(* Schneider Machine Expert - Basic project automat_biscuiti, file version 2.6.0.0 *)
(* ProjectInformations: Name=New project *)

HARDWARE
  Cpu 0: TM221M16R/G
  ModuleExtensionObject 0: TM3AM6/G
  ModuleExtensionObject 1: TM3AI8/G
  EthernetConfiguration: NetworkName=M221, IpAllocationMode=FixedAddress, IpAddress=0.0.0.0, SubnetMask=0.0.0.0
  SerialLineConfiguration: Baud=Baud19200, Parity=ParityEven, DataBits=DataBits8, StopBits=StopBits1, PhysicalMedium=PhysicalMediumRs485, TransmissionMode=TransmissionModeModbusRtu, SlaveId=1, Addressing=SlaveAddressing
  MastTask: UsePeriodScanMode=false, PeriodScan=100
  FastTask: Period=255
  CpuBehavior: StartingMode=StartAsPreviousState, AutoSaveRamOnEeprom=true, WatchdogPeriod=250

SYMBOLS  (address, symbol, comment, settings)
  %TM0        "Se pregatesc biscuitii"  [Preset=5, Base=OneSecond]
  %I0.0       "Faina fara gluten"
  %I0.1       "Faina integrala"
  %I0.2       "Lapte"
  %I0.3       "Lapte de soia"
  %I0.4       "Lapte de migdale"
  %I0.5       "Ou"
  %I0.6       "Inlocuitor ou"
  %I0.7       "Automat pornit"
  %Q0.0       "Faina fara gluten"
  %Q0.1       "Faina integrala"
  %Q0.2       "Lapte"
  %Q0.3       "Lapte de soia"
  %Q0.4       "Automat pornit - introduceti 15 lei"
  %Q0.5       "Ou"
  %Q0.6       "Inlocuitor ou"
  %Q0.7       "Cutie biscuiti servita"
  %IW0.0      [Type=Type_0_10V, Scope=Scope_Normal, Minimum=0, Maximum=1000]
  %IW1.1      [Type=Type_NotUsed, Scope=Scope_NotUsed, Minimum=0, Maximum=0]

POU New POU
  (* SectionNumber=1 *)

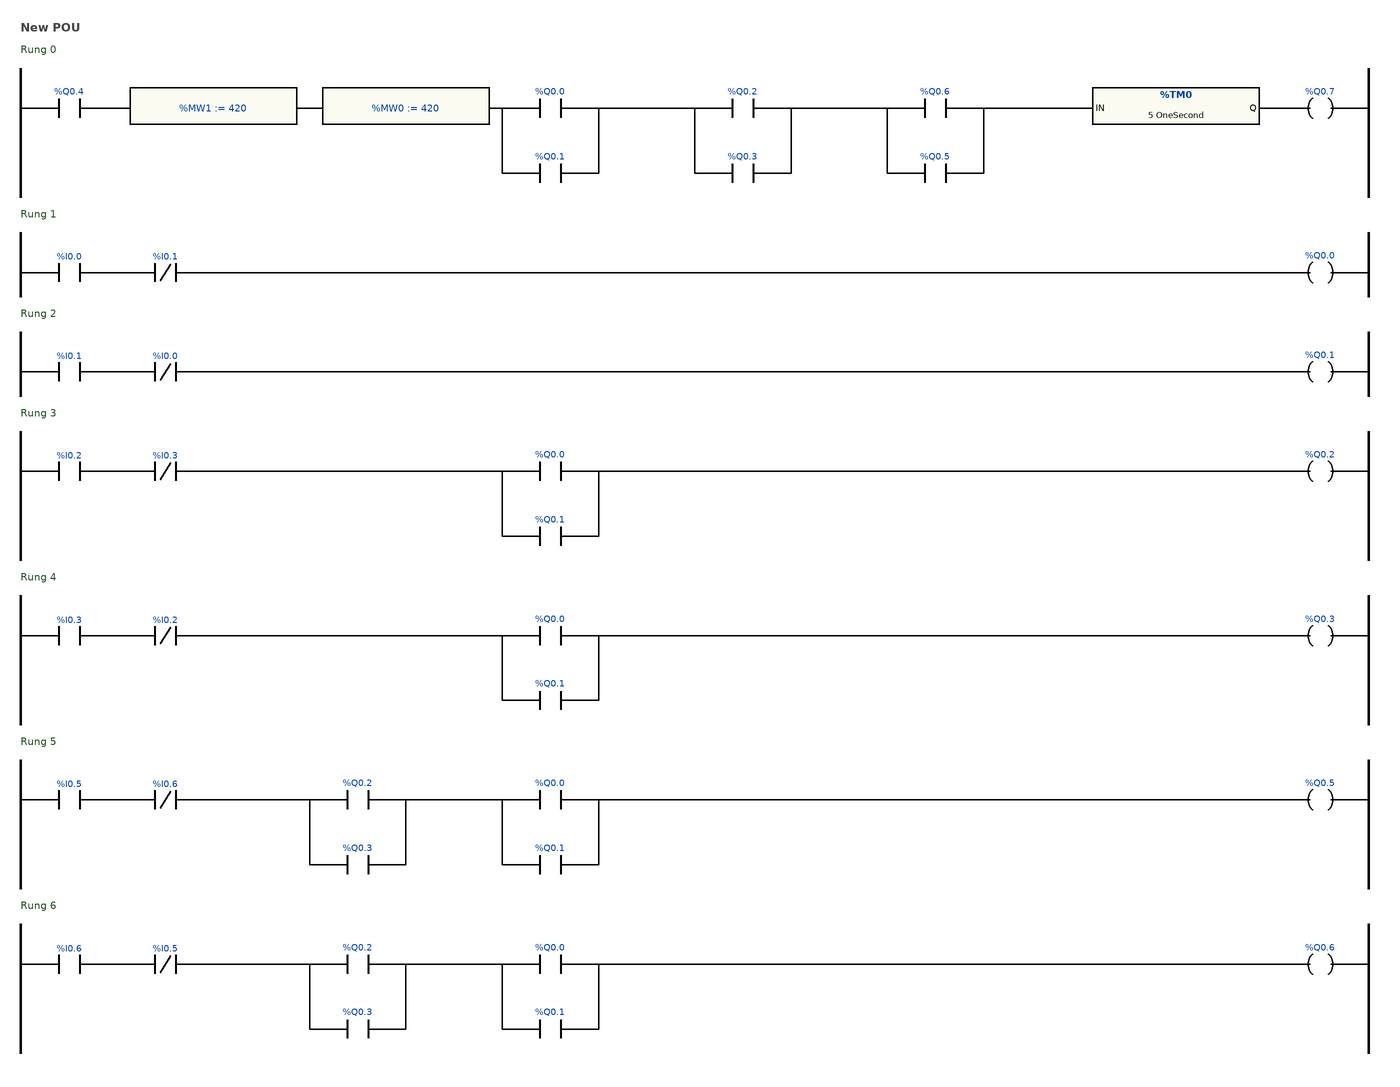

// Rung 0
  BLK %TM0
  LD %Q0.4
  OPER [ %MW1 := 420 ]
  OPER [ %MW0 := 420 ]
  AND( %Q0.0
  OR %Q0.1
  )
  AND( %Q0.2
  OR %Q0.3
  )
  AND( %Q0.6
  OR %Q0.5
  )
  IN
  OUT_BLK
  LD Q
  ST %Q0.7
  END_BLK
  // as ST:
  //   IF %Q0.4 THEN %MW1 := 420; END_IF;
  //   IF %Q0.4 THEN %MW0 := 420; END_IF;
  //   %TM0(IN := %Q0.4 AND (%Q0.0 OR %Q0.1) AND (%Q0.2 OR %Q0.3) AND (%Q0.6 OR %Q0.5));
  //   %Q0.7 := %TM0.Q;

// Rung 1
  LD %I0.0
  ANDN %I0.1
  ST %Q0.0
  // as ST:
  //   %Q0.0 := %I0.0 AND NOT %I0.1;

// Rung 2
  LD %I0.1
  ANDN %I0.0
  ST %Q0.1
  // as ST:
  //   %Q0.1 := %I0.1 AND NOT %I0.0;

// Rung 3
  LD %I0.2
  ANDN %I0.3
  AND( %Q0.0
  OR %Q0.1
  )
  ST %Q0.2
  // as ST:
  //   %Q0.2 := %I0.2 AND NOT %I0.3 AND (%Q0.0 OR %Q0.1);

// Rung 4
  LD %I0.3
  ANDN %I0.2
  AND( %Q0.0
  OR %Q0.1
  )
  ST %Q0.3
  // as ST:
  //   %Q0.3 := %I0.3 AND NOT %I0.2 AND (%Q0.0 OR %Q0.1);

// Rung 5
  LD %I0.5
  ANDN %I0.6
  AND( %Q0.2
  OR %Q0.3
  )
  AND( %Q0.0
  OR %Q0.1
  )
  ST %Q0.5
  // as ST:
  //   %Q0.5 := %I0.5 AND NOT %I0.6 AND (%Q0.2 OR %Q0.3) AND (%Q0.0 OR %Q0.1);

// Rung 6
  LD %I0.6
  ANDN %I0.5
  AND( %Q0.2
  OR %Q0.3
  )
  AND( %Q0.0
  OR %Q0.1
  )
  ST %Q0.6
  // as ST:
  //   %Q0.6 := %I0.6 AND NOT %I0.5 AND (%Q0.2 OR %Q0.3) AND (%Q0.0 OR %Q0.1);

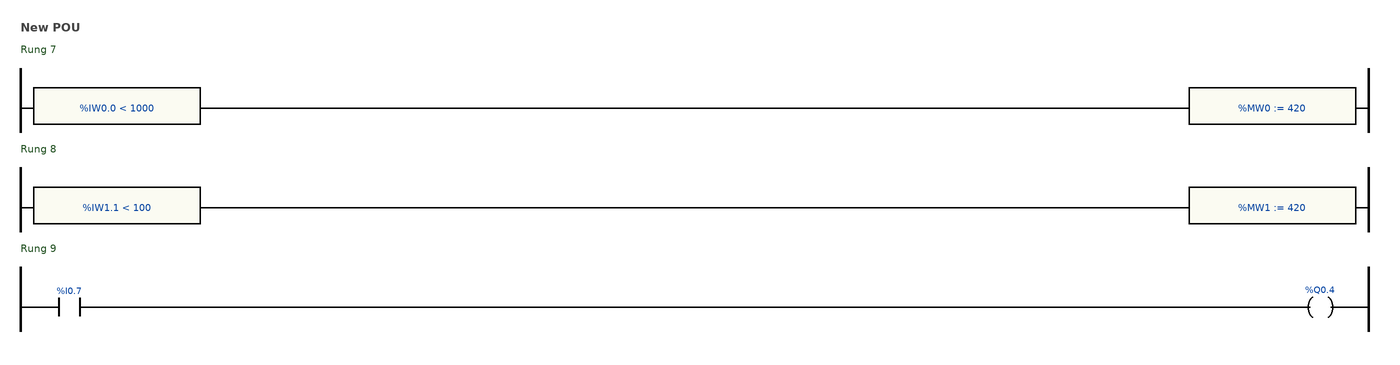

// Rung 7
  LD [ %IW0.0 < 1000 ]
  [ %MW0 := 420 ]
  // as ST:
  //   IF %IW0.0 < 1000 THEN %MW0 := 420; END_IF;

// Rung 8
  LD [ %IW1.1 < 100 ]
  [ %MW1 := 420 ]
  // as ST:
  //   IF %IW1.1 < 100 THEN %MW1 := 420; END_IF;

// Rung 9
  LD %I0.7
  ST %Q0.4
  // as ST:
  //   %Q0.4 := %I0.7;
